FUNCTION_BLOCK "FB_Sensor"
TITLE = FB_PEC
{ S7_Optimized_Access := 'TRUE' }
AUTHOR : MHSE
FAMILY : Conveyor
VERSION : 3.0
// ATTRIBUTES
// AUTO_NUMBER = True
// BLOCK_NUMBER = 219
// END_ATTRIBUTES
   VAR_INPUT
      ix_PEC { ExternalAccessible := 'False'; ExternalVisible := 'False'; ExternalWritable := 'False'} : Bool;   // Signal of the PEC
      iUDT_PECConfiguration { ExternalAccessible := 'False'; ExternalVisible := 'False'; ExternalWritable := 'False'} : "UDT_PECConfiguration";   // PEC configuration structure
   END_VAR

   VAR_OUTPUT
      qx_PECFiltered { ExternalAccessible := 'False'; ExternalVisible := 'False'; ExternalWritable := 'False'} : Bool;   // PEC Filtered
      qUDT_HMIStatus { ExternalAccessible := 'False'; ExternalVisible := 'False'; ExternalWritable := 'False'} : "UDT_PECStatus";   // Status structure
   END_VAR

   VAR_IN_OUT
      iqUDT_ConveyorInterface : "UDT_ConveyorInterface";   // Interface structure
      iqUDT_PECStatistics : "UDT_PECStatistics";   // Statistics structure
   END_VAR

   VAR
      s_Status { ExternalAccessible := 'False'; ExternalVisible := 'False'; ExternalWritable := 'False'; S7_SetPoint := 'False'} : "UDT_PECStatus";   // Status structure
      s_StatusOld { ExternalAccessible := 'False'; ExternalVisible := 'False'; ExternalWritable := 'False'; S7_SetPoint := 'False'} : "UDT_PECStatus";   // Auxiliary status structure
      sx_Enable { ExternalAccessible := 'False'; ExternalVisible := 'False'; ExternalWritable := 'False'} : Bool;   // Enable
   END_VAR
   VAR RETAIN
      si_AuxJamDisplacement { ExternalAccessible := 'False'; ExternalVisible := 'False'; ExternalWritable := 'False'} : Int;   // Auxiliary variable to calculate displacement when PEC is blocked
   END_VAR
   VAR
      sx_PECFiltered { ExternalAccessible := 'False'; ExternalVisible := 'False'; ExternalWritable := 'False'} : Bool;   // Photo eye filtered
      PEC_TimerOnOffDelay { ExternalAccessible := 'False'; ExternalVisible := 'False'; ExternalWritable := 'False'; S7_SetPoint := 'False'} : "FB_TimerOnOffDelay";   // Filtering end of section photo eye signal
      R_TRIG_PECJam {InstructionName := 'R_TRIG'; LibVersion := '1.0'; ExternalAccessible := 'False'; ExternalVisible := 'False'; ExternalWritable := 'False'; S7_SetPoint := 'False'} : R_TRIG;   // Rising edge trigger PEC jam
   END_VAR


BEGIN
	(*
	----------------------------------------------------------------------------------------

	Version history:
	Date        | Version   | Author        | Remark
	----------------------------------------------------------------------------------------
	04/10/2019  | 2.0       | S. Nikodem    | first release TIA 15.1
	09/10/2019  | 2.1       | L.Klar        | Internal PEC error added
	28/10/2019  | 2.2       | S. Nikodem    | Change sign in region 2 - equal to greater then
	29/10/2019  | 2.3       | L.Klar        | UDT_PECStatus output variable changed, interface comments adjusted
	29/10/2019  | 2.4       | L.Klar        | Region 4 - time input corrected
	12/11/2019  | 3.0       | P.Majka       | 3.0 MHS library release TIA 15.1
	26/11/2019  | 3.1       | P.Majka       | Static variable name change to PEC from EOS PEC
	12/12/2019  | 3.2       | C. Leite      | Absolute displacement value to control jam error in both directions
	21/02/2023  | 4.0       | F.Baten       | 4.0 Release TIA 17.5
	12/03/2024  | 4.1       | S. Nieswiec   | Small variable name changes according to current standard
	*)

	REGION 1 - Triggers

	    // Rising edge PEC Jam
	    #R_TRIG_PECJam(CLK := #s_Status.Jam);

	END_REGION

	REGION 2 - Active function

	    // To activate the jam monitoring the jam displacement limit  must be configured up to zero.
	    #sx_Enable := #iUDT_PECConfiguration.JamDisplacementLimit > 0;

	END_REGION

	REGION 3 - Reset errors

	    // Jam error is reset when reset bit is active and jam error is active and is connfigured alllow reset jam with PEC blocked or photo eye is not active
	    IF #iqUDT_ConveyorInterface.InternalErrorReset
	        AND (#iUDT_PECConfiguration.ResetWithPECBlocked
	        OR (NOT #iUDT_PECConfiguration.ResetWithPECBlocked
	        AND #sx_PECFiltered))
	        AND #s_Status.Jam
	    THEN

	        #si_AuxJamDisplacement := 0;
	        #s_Status.Jam := FALSE;

	    END_IF;

	END_REGION

	REGION 4 - Photo eye filters

	    // End of section photo eye signal filter timer
	    #PEC_TimerOnOffDelay(iudi_OnDelayTime := #iUDT_PECConfiguration.TimeOnDelay,
	                         iudi_OffDelayTime := #iUDT_PECConfiguration.TimeOffDelay,
	                         ix_SignalToDelay := #ix_PEC,
	                         ix_Enable := TRUE,
	                         qx_DelayedSignal => #sx_PECFiltered);

	    // Write the current status of the photo eye
	    #s_Status.PEC := #sx_PECFiltered;
	    #qx_PECFiltered := #sx_PECFiltered;

	END_REGION

	REGION 5 - Jam detection

	    IF NOT #sx_PECFiltered                                                    // Photo eye blocked
	        AND #sx_Enable                                                            // Active of checking the PEC jam
	    THEN

	        #si_AuxJamDisplacement += ABS(#iqUDT_ConveyorInterface.Displacement);

	    ELSE

	        #si_AuxJamDisplacement := 0;

	    END_IF;

	    // Compare jam auxiliary counter with displacement jam configured
	    IF #si_AuxJamDisplacement > #iUDT_PECConfiguration.JamDisplacementLimit
	    THEN

	        #s_Status.Jam := TRUE;

	    END_IF;

	END_REGION

	REGION 6 - Statistics

	    // Statistics Jam PEC
	    IF #s_Status.Jam                                                                // PEC jam error active
	        OR #iqUDT_ConveyorInterface.ResetStatistics                                       // Reset statistics
	    THEN

	        "FC_Statistics"(ix_Reset := #iqUDT_ConveyorInterface.ResetStatistics,
	                        ix_Activate := #s_Status.Jam,
	                        ix_RTrigActivate := #R_TRIG_PECJam.Q,
	                        iqUDT_Statistics := #iqUDT_PECStatistics.Jam);

	    END_IF;

	END_REGION

	REGION 7 - Internal PEC error

	    IF #s_Status.Jam
	    THEN

	        #iqUDT_ConveyorInterface.InternalErrorPEC := TRUE;

	    END_IF;

	END_REGION


	REGION 8 - Status

	    // Status update on change
	    IF #s_StatusOld <> #s_Status
	    THEN

	        #qUDT_HMIStatus := #s_Status;
	        #s_StatusOld := #s_Status;

	    END_IF;

	END_REGION
END_FUNCTION_BLOCK

